ABB RobotStudio station: EstacionTaladrado_20230526-132759.rsstn

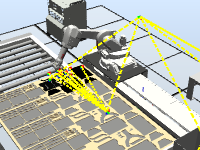
Station EstacionTaladrado (saved by RobotStudio 6.8.8307.1040)
Controller IRB1600APM, task T_ROB2: task frame (RAPID world) sits at (108, -1423.5, 460) mm, rotated rx 0 ry 0 rz 90 deg in the station
Controller IRB1600APM, task T_ROB1: task frame (RAPID world) sits at (108, -1423.5, 460) mm, rotated rx 0 ry 0 rz 90 deg in the station
Controller IRB1600APM
  mechanical unit ROB_1: IRB1600_6_145_A, 6 joints, base frame (0, 0, 0) mm
  mechanical unit TRACK_1: IRBT2005_IRB_STD_INT_0_0_4_A, 1 joints, base frame (0, 0, 0) mm
  mechanical unit ROB_2: IRB1600_6_145_B, 6 joints, base frame (1847, 2866, 0) mm, rotated rx 0 ry 0 rz 180 deg
  mechanical unit TRACK_2: IRBT2005_IRB_STD_INT_0_0_4_B, 1 joints, base frame (1847, 2866, 0) mm, rotated rx 0 ry 0 rz 180 deg
Layout (positions relative to the parent item):
  - Placa_de_Corte [part] at (-2250, -1220, 450) mm
  - IRC5_Singel-Cabinet [part, from Equipment\IRC5_Singel-Cabinet.rslib] at (500, 3000, 100) mm, rotated rx 90 ry 0 rz 90 deg
  - 1320_4000_h2 [part, from Equipment\Conveyor 1320 4000 h2.rslib] at (-1985, 2800, 0) mm, rotated rx 0 ry 0 rz -90 deg
  - Ventosa_Smart [smart component]
      signals: DI StartAttacher, DO Executed
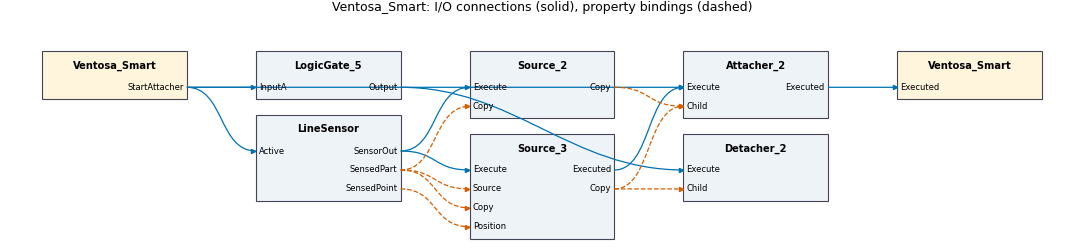
      connections:
        Ventosa_Smart.StartAttacher -> LogicGate_5.InputA
        LogicGate_5.Output -> Detacher_2.Execute
        Ventosa_Smart.StartAttacher -> LineSensor.Active
        Ventosa_Smart.StartAttacher -> Attacher_2.Execute
        Attacher_2.Executed -> Ventosa_Smart.Executed
        LineSensor.SensorOut -> Source_2.Execute
        LineSensor.SensorOut -> Source_3.Execute
        Source_3.Executed -> Attacher_2.Execute
        LineSensor.SensedPart => Source_2.Copy
        Source_2.Copy => Attacher_2.Child
        LineSensor.SensedPart => Source_3.Source
        LineSensor.SensedPart => Source_3.Copy
        Source_3.Copy => Attacher_2.Child
        Source_3.Copy => Detacher_2.Child
        LineSensor.SensedPoint => Source_3.Position
    - Attacher_2 [smart component, from Components\Attacher.rslib]
        properties: Parent=Ventosa; Flange=0; Child=(none); Mount=false; Offset=[0 0 0]; Orientation=[0 0 0]
    - Detacher_2 [smart component, from Components\Detacher.rslib]
        properties: Child=(none); KeepPosition=true
    - LogicGate_5 [smart component, from Components\LogicGate.rslib]
        properties: Operator=NOT; Delay=0
    - LineSensor [smart component, from Components\LineSensor.rslib] at (-959.44, 1157.84, 473.42) mm, rotated rx -180 ry 0 rz 0 deg
        properties: Start=[0 0 0]; End=[6.66133814775094E-16 -4.71844785465692E-16 0.00999998807907376]; Radius=0.006; SensedPart=(none); SensedPoint=[0 0 0]
      - _sensorPart_ [part]
    - Ventosa [mechanism, from Libraries\Ventosa.rslib] at (-959.44, 1157.84, 583.42) mm, rotated rx -180 ry 0 rz 0 deg
    - Source_3 [smart component, from Components\Source.rslib]
        properties: Source=(none); Copy=(none); Parent=(none); Position=[0 0 0]; Orientation=[0 0 0]; Transient=false; PhysicsBehavior=0
  - PLACA_SOPORTE_1 [part] at (-1200.46, 988.98, 450) mm
  - BANDEJA_LAMINA [part]
  - MyTool [mechanism, from Training Objects\myTool.rslib] at (-2758, -382.79, 1614) mm, rotated rx 180 ry 60 rz 90 deg
  - SOPORTE_LATERAL_SOPORTE_1 [part] at (-961.81, 1075.54, 450) mm
  - MESA_TALADRADO [part] at (1200, -425, 400) mm
  - MESA_TALADRADO_B [part] at (-3850, 0, 400) mm
  - IRB1600_6_145_A [mechanism, from Robots\IRB1600_6_145_G_02.rslib] at (108, 926.5, 460) mm, rotated rx 0 ry 0 rz 90 deg; joint values [1.3574, 1.2334, -0.1513, 0, 0.4887, -0.2134] (rad or m)
  - IRB1600_6_145_B [mechanism, from Robots\IRB1600_6_145_G_02.rslib] at (-2758, 423.5, 460) mm, rotated rx 0 ry 0 rz -90 deg; joint values [0, 0, 0, 0, 0.5236, 0] (rad or m)
  - IRBT2005_IRB_STD_INT_0_0_4_A [mechanism] at (400, -2248, 0) mm, rotated rx 0 ry 0 rz 90 deg; joint values [2.35] (rad or m)
      links: Base, Link1
  - IRBT2005_IRB_STD_INT_0_0_4_B [mechanism] at (-3050, 1248, 0) mm, rotated rx 0 ry 0 rz -90 deg; joint values [0] (rad or m)
      links: Base, Link1
  - Conveyor_A [smart component]
      signals: DI MoveConv
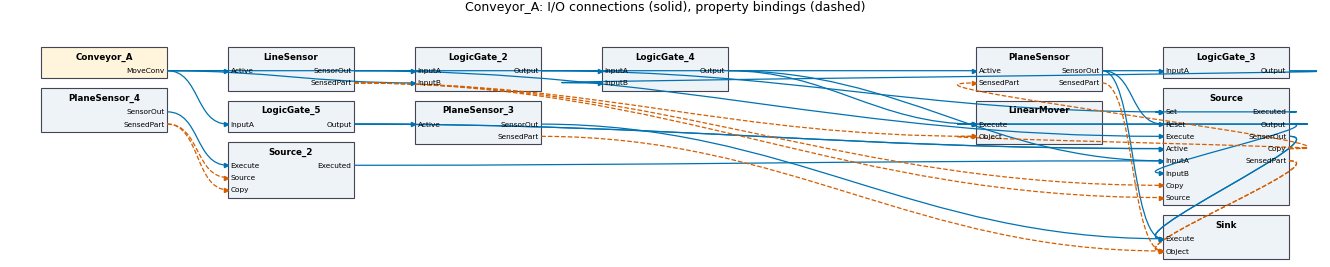
      connections:
        Source.Executed -> LogicSRLatch.Set
        PlaneSensor.SensorOut -> LogicSRLatch.Reset
        Conveyor_A.MoveConv -> LineSensor.Active
        LineSensor.SensorOut -> Source.Execute
        LogicSRLatch.Output -> LinearMover.Execute
        Conveyor_A.MoveConv -> PlaneSensor.Active
        LineSensor.SensorOut -> LogicGate_2.InputA
        Conveyor_A.MoveConv -> LogicGate_2.InputB
        LogicGate_2.Output -> LogicSRLatch.Set
        PlaneSensor.SensorOut -> LogicGate_3.InputA
        LogicGate_2.Output -> LogicGate_4.InputA
        LogicGate_3.Output -> LogicGate_4.InputB
        PlaneSensor.SensorOut -> Sink.Execute
        PlaneSensor_2.SensorOut -> Sink.Execute
        Conveyor_A.MoveConv -> LogicGate_5.InputA
        LogicGate_5.Output -> PlaneSensor_2.Active
        LogicGate_5.Output -> LineSensor.Active
        LineSensor.SensorOut -> Sink.Execute
        PlaneSensor_3.SensorOut -> Sink.Execute
        LogicGate_5.Output -> PlaneSensor_3.Active
        PlaneSensor_4.SensorOut -> Source_2.Execute
        LogicGate_4.Output -> LogicGate_8.InputA
        LogicGate_8.Output -> LinearMover.Execute
        LogicGate_9.Output -> LogicGate_8.InputB
        Source_2.Executed -> LogicGate_9.InputA
        LogicGate_4.Output -> LinearMover.Execute
        LineSensor.SensedPart => Source.Copy
        Source.Copy => LinearMover.Object
        Source.Copy => PlaneSensor.SensedPart
        LineSensor.SensedPart => Source.Source
        PlaneSensor_2.SensedPart => Sink.Object
        LineSensor.SensedPart => Sink.Object
        PlaneSensor_3.SensedPart => Sink.Object
        LineSensor.SensedPart => LinearMover.Object
        PlaneSensor.SensedPart => Sink.Object
        PlaneSensor_4.SensedPart => Source_2.Source
        PlaneSensor_4.SensedPart => Source_2.Copy
    - PlaneSensor [smart component, from Components\PlaneSensor.rslib]
        properties: Origin=[-1.025 -4.3 0.776]; Axis1=[0 0 0.099]; Axis2=[0.39 0 0]; SensedPart=(none)
      - _sensorPart_ [part]
    - LineSensor [smart component, from Components\LineSensor.rslib]
        properties: Start=[-0.83 -1.7 0.78]; End=[-0.83 -4.3 0.785]; Radius=0.005; SensedPart=BOX_A; SensedPoint=[-0.83 -1.7 0.78]
      - _sensorPart_ [part]
    - LinearMover [smart component, from Components\LinearMover.rslib]
        properties: Object=BOX_A; Direction=[0 -3.5 0]; Speed=0.5; Reference=Global; ReferenceObject=(none)
    - LogicGate_2 [smart component, from Components\LogicGate.rslib]
        properties: Operator=AND; Delay=0
    - LogicGate_3 [smart component, from Components\LogicGate.rslib]
        properties: Operator=NOT; Delay=0
    - LogicGate_4 [smart component, from Components\LogicGate.rslib]
        properties: Operator=AND; Delay=0
    - Sink [smart component, from Components\Sink.rslib]
        properties: Object=(none)
    - LogicGate_5 [smart component, from Components\LogicGate.rslib]
        properties: Operator=NOT; Delay=0
    - PlaneSensor_3 [smart component, from Components\PlaneSensor.rslib]
        properties: Origin=[-1.02 -2 0.786]; Axis1=[0.38 0 0]; Axis2=[0 0.3 0]; SensedPart=(none)
      - _sensorPart_ [part]
    - Source_2 [smart component, from Components\Source.rslib]
        properties: Source=(none); Copy=(none); Parent=(none); Position=[-0.83 -1.85 0.776]; Orientation=[0 0 0]; Transient=false; PhysicsBehavior=0
    - PlaneSensor_4 [smart component, from Components\PlaneSensor.rslib]
        properties: Origin=[-1.025 -4.3 0.776]; Axis1=[0 0 0.099]; Axis2=[0.39 0 0]; SensedPart=(none)
      - _sensorPart_ [part]
  - 400_guide_B [part, from Equipment\Conveyor Guide 400.rslib] at (-1955, -1500, 0) mm, rotated rx 0 ry 0 rz -90 deg
  - 400_guide_A [part, from Equipment\Conveyor Guide 400.rslib] at (-1030, -1500, 0) mm, rotated rx 0 ry 0 rz -90 deg
  - SOPORTE_LATERAL_SOPORTE_1_2 [part] at (-1011.44, 1038.99, 450) mm
  - BASE_SOPORTE_1 [part] at (-878.76, 996.15, 450) mm
  - GRADUADOR_INCLINACION_SOPORTE_1 [part] at (-1023.59, 997.95, 450) mm
  - GRADUADOR_INCLINACION_SOPORTE_1_2 [part] at (-966.4, 1160.33, 450) mm
  - SUJECION_CENTRAL_SOPORTE_1 [part] at (-870.47, 885.99, 450) mm
  - BRAZO_SOPORTE_1 [part] at (-762.24, 1077.84, 450) mm
  - BRAZO_2_SOPORTE_1 [part] at (-1135.46, 1150.12, 450) mm
  - BOX_A [part] at (-830, -1850, 776) mm
  - PLACA_INFERIOR_MESA_1 [part] at (-558.01, 1007.22, 450) mm
  - PLACA_SUPERIOR_MESA_1 [part] at (-913.92, 730.48, 450) mm
  - SOPORTE_LATERAL_I_MESA_1 [part] at (-1245.6, 782.8, 450) mm
  - SOPORTE_LATERAL_D_MESA_1 [part] at (-580.16, 719.3, 450) mm
Attachment: LineSensor is attached to Ventosa / HERRAMIENTA
Attachment: Ventosa is attached to IRB1600_6_145_A / Link6
Attachment: MyTool is attached to IRB1600_6_145_B / Link6
Attachment: IRB1600_6_145_A is attached to IRBT2005_IRB_STD_INT_0_0_4_A / Link1
Attachment: IRB1600_6_145_B is attached to IRBT2005_IRB_STD_INT_0_0_4_B / Link1
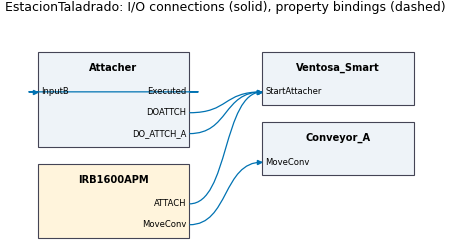
Station logic (signal -> signal, property => property):
  Attacher.Executed -> LogicGate.InputB
  IRB1600APM.DOATTCH -> Ventosa_Smart.StartAttacher
  IRB1600APMSYS.DO_ATTCH_A -> Ventosa_Smart.StartAttacher
  IRB1600APM.ATTACH -> Ventosa_Smart.StartAttacher
  IRB1600APM.MoveConv -> Conveyor_A.MoveConv
Targets, tools, work objects and paths stored in the station, written as RAPID:
! task T_ROB1
MODULE CalibData
  PERS tooldata VentosaTCP:=[TRUE,[[0,0,110.772],[1,0,0,0]],[1,[0,0,53.582],[1,0,0,0],0,0,0]];
  TASK PERS wobjdata PLACA_A:=[FALSE,TRUE,"",[[0,0,0],[1,0,0,0]],[[203.5,2358,-10],[0.707106781,0,0,-0.707106781]]];
ENDMODULE

! task T_ROB1
MODULE Module1
  CONST jointtarget HOME_A:=[[0,0,0,0,30,0],[925,9E+09,9E+09,9E+09,9E+09,9E+09]];
  CONST jointtarget MID_A:=[[90,60,-20,0,50,0],[925,9E+09,9E+09,9E+09,9E+09,9E+09]];
  CONST jointtarget TABLE_A:=[[-86.149,71.536,-9.408,0,27.873,0],[925,9E+09,9E+09,9E+09,9E+09,9E+09]];
  CONST jointtarget SLS1_A:=[[82.069,70.996,-7.558,0,26.562,0],[2350,9E+09,9E+09,9E+09,9E+09,9E+09]];
  CONST jointtarget PS1_A:=[[87.22,84.052,-44.6,0,50.548,0],[2349.769019747,9E+09,9E+09,9E+09,9E+09,9E+09]];
  CONST jointtarget PS1_AA:=[[87.22,83.446,-44.115,0,50.669,0],[2349.769019747,9E+09,9E+09,9E+09,9E+09,9E+09]];
  CONST jointtarget PSLS1_AA:=[[82.069,69.527,-6.738,0,27.211,0],[2350,9E+09,9E+09,9E+09,9E+09,9E+09]];
  CONST jointtarget CONVEYOR_A:=[[84.914,41.92,15.328,-0.622,32.813,0],[-461.181385797,9E+09,9E+09,9E+09,9E+09,9E+09]];
  CONST jointtarget MID_CONV_A:=[[89.175,20.381,4.444,0.004,65.253,0],[-480,9E+09,9E+09,9E+09,9E+09,9E+09]];
  CONST jointtarget SLS12_AA:=[[84.262,72.054,-13.066,0,31.013,0],[2350,9E+09,9E+09,9E+09,9E+09,9E+09]];
  CONST jointtarget SLS12_A:=[[84.105,72.802,-13.543,0,30.74,0],[2350,9E+09,9E+09,9E+09,9E+09,9E+09]];
  CONST jointtarget BS1_A:=[[84.635,68.196,3.223,0,18.581,0],[2350,9E+09,9E+09,9E+09,9E+09,9E+09]];
  CONST jointtarget BS1_AA:=[[84.635,67.383,3.658,0,18.96,0],[2350,9E+09,9E+09,9E+09,9E+09,9E+09]];
  CONST jointtarget GIS1_AA:=[[86.51,72.134,-13.296,0,31.162,0],[2350,9E+09,9E+09,9E+09,9E+09,9E+09]];
  CONST jointtarget GIS1_A:=[[86.51,72.86,-13.724,0,30.865,0],[2350,9E+09,9E+09,9E+09,9E+09,9E+09]];
  CONST jointtarget GIS12_AA:=[[77.771,70.671,-8.671,0,28,0],[2350,9E+09,9E+09,9E+09,9E+09,9E+09]];
  CONST jointtarget GIS12_A:=[[77.79,71.449,-9.107,0,27.659,0],[2350,9E+09,9E+09,9E+09,9E+09,9E+09]];
  CONST jointtarget BRS1_A:=[[80.135,66.069,14.969,0,8.962,0],[2350,9E+09,9E+09,9E+09,9E+09,9E+09]];
  CONST jointtarget BRS1_AA:=[[80.135,65.237,15.395,0,9.368,0],[2350,9E+09,9E+09,9E+09,9E+09,9E+09]];
  CONST jointtarget BRS12_A:=[[79.805,80.411,-35.266,0,44.855,0],[2350,9E+09,9E+09,9E+09,9E+09,9E+09]];
  CONST jointtarget BRS12_AA:=[[79.805,79.69,-34.75,0,45.061,0],[2350,9E+09,9E+09,9E+09,9E+09,9E+09]];
  CONST jointtarget SCS1_A:=[[92.371,67.896,4.57,0,17.533,0],[2350,9E+09,9E+09,9E+09,9E+09,9E+09]];
  CONST jointtarget SCS1_AA:=[[92.371,67.108,4.99,0,17.903,0],[2350,9E+09,9E+09,9E+09,9E+09,9E+09]];
  CONST jointtarget PIM1_A:=[[56.022,65.432,22.991,0,1.578,0],[1981.865508797,9E+09,9E+09,9E+09,9E+09,9E+09]];
  CONST jointtarget PIM1_AA:=[[56.022,64.534,23.445,0,2.021,0],[1981.865508797,9E+09,9E+09,9E+09,9E+09,9E+09]];
  CONST jointtarget TABLE_AA:=[[-86.149,55.011,-3.204,0,38.193,0],[925,9E+09,9E+09,9E+09,9E+09,9E+09]];
  CONST jointtarget TABLE_A90:=[[-86.149,55.011,-3.204,0,38.193,90],[925,9E+09,9E+09,9E+09,9E+09,9E+09]];
  CONST jointtarget TABLE_A180:=[[-86.149,55.011,-3.204,0,38.193,180],[925,9E+09,9E+09,9E+09,9E+09,9E+09]];
  CONST jointtarget TABLE_A270:=[[-86.149,55.011,-3.204,0,38.193,270],[925,9E+09,9E+09,9E+09,9E+09,9E+09]];
  PROC Path_HOME_A()
    MoveAbsJ HOME_A,v1000,z100,VentosaTCP\WObj:=PLACA_A;
  ENDPROC
  PROC Path_MID_A()
    MoveAbsJ MID_A,v1000,z100,VentosaTCP\WObj:=PLACA_A;
  ENDPROC
  PROC Path_PS1_A()
    MoveAbsJ PS1_A,v1000,z100,VentosaTCP\WObj:=PLACA_A;
    MoveAbsJ PS1_AA,v1000,z100,VentosaTCP\WObj:=PLACA_A;
    MoveAbsJ HOME_A,v1000,z100,VentosaTCP\WObj:=PLACA_A;
    MoveAbsJ MID_CONV_A,v1000,z100,VentosaTCP\WObj:=PLACA_A;
    MoveAbsJ CONVEYOR_A,v1000,z100,VentosaTCP\WObj:=PLACA_A;
  ENDPROC
  PROC Path_PS1_AA()
    MoveAbsJ PS1_AA,v1000,z100,VentosaTCP\WObj:=PLACA_A;
  ENDPROC
  PROC Path_MID_CONV_A()
    MoveAbsJ MID_CONV_A,v1000,z100,VentosaTCP\WObj:=PLACA_A;
  ENDPROC
  PROC Path_SLS1_A()
    MoveAbsJ SLS1_A,v1000,z100,VentosaTCP\WObj:=PLACA_A;
    MoveAbsJ PSLS1_AA,v1000,z100,VentosaTCP\WObj:=PLACA_A;
    MoveAbsJ MID_A,v1000,z100,VentosaTCP\WObj:=PLACA_A;
    MoveAbsJ HOME_A,v1000,z100,VentosaTCP\WObj:=PLACA_A;
    MoveAbsJ TABLE_A,v1000,z100,VentosaTCP\WObj:=PLACA_A;
  ENDPROC
  PROC Path_SLS1_AA()
    MoveAbsJ PSLS1_AA,v1000,z100,VentosaTCP\WObj:=PLACA_A;
  ENDPROC
  PROC Path_SLS12_AA()
    MoveAbsJ SLS12_AA,v1000,z100,VentosaTCP\WObj:=PLACA_A;
  ENDPROC
  PROC Path_SLS12_A()
    MoveAbsJ SLS12_A,v1000,z100,VentosaTCP\WObj:=PLACA_A;
    MoveAbsJ SLS12_AA,v1000,z100,VentosaTCP\WObj:=PLACA_A;
    MoveAbsJ MID_A,v1000,z100,VentosaTCP\WObj:=PLACA_A;
    MoveAbsJ HOME_A,v1000,z100,VentosaTCP\WObj:=PLACA_A;
    MoveAbsJ TABLE_A,v1000,z100,VentosaTCP\WObj:=PLACA_A;
  ENDPROC
  PROC Path_BS1_A()
    MoveAbsJ BS1_A,v1000,z10,VentosaTCP\WObj:=PLACA_A;
    MoveAbsJ BS1_AA,v1000,z10,VentosaTCP\WObj:=PLACA_A;
    MoveAbsJ MID_A,v1000,z10,VentosaTCP\WObj:=PLACA_A;
    MoveAbsJ HOME_A,v1000,z10,VentosaTCP\WObj:=PLACA_A;
    MoveAbsJ MID_CONV_A,v1000,z10,VentosaTCP\WObj:=PLACA_A;
    MoveAbsJ CONVEYOR_A,v1000,z10,VentosaTCP\WObj:=PLACA_A;
  ENDPROC
  PROC Path_BS1_AA()
    MoveAbsJ BS1_AA,v1000,z10,VentosaTCP\WObj:=PLACA_A;
  ENDPROC
  PROC Path_SLS1_A_2()
    MoveAbsJ HOME_A,v1000,z100,VentosaTCP\WObj:=PLACA_A;
    MoveAbsJ MID_CONV_A,v1000,z100,VentosaTCP\WObj:=PLACA_A;
    MoveAbsJ CONVEYOR_A,v1000,z100,VentosaTCP\WObj:=PLACA_A;
  ENDPROC
  PROC Path_SLS12_A_2()
    MoveAbsJ HOME_A,v1000,z100,VentosaTCP\WObj:=PLACA_A;
    MoveAbsJ MID_CONV_A,v1000,z100,VentosaTCP\WObj:=PLACA_A;
    MoveAbsJ CONVEYOR_A,v1000,z100,VentosaTCP\WObj:=PLACA_A;
  ENDPROC
  PROC Path_GIS1_A()
    MoveAbsJ GIS1_A,v1000,z10,VentosaTCP\WObj:=PLACA_A;
    MoveAbsJ GIS1_AA,v1000,z10,VentosaTCP\WObj:=PLACA_A;
    MoveAbsJ MID_A,v1000,z10,VentosaTCP\WObj:=PLACA_A;
    MoveAbsJ HOME_A,v1000,z10,VentosaTCP\WObj:=PLACA_A;
    MoveAbsJ TABLE_A,v1000,z10,VentosaTCP\WObj:=PLACA_A;
  ENDPROC
  PROC Path_GIS1_AA()
    MoveAbsJ GIS1_AA,v1000,z10,VentosaTCP\WObj:=PLACA_A;
  ENDPROC
  PROC Path_GIS1_A_2()
    MoveAbsJ HOME_A,v1000,z10,VentosaTCP\WObj:=PLACA_A;
    MoveAbsJ MID_CONV_A,v1000,z10,VentosaTCP\WObj:=PLACA_A;
    MoveAbsJ CONVEYOR_A,v1000,z10,VentosaTCP\WObj:=PLACA_A;
  ENDPROC
  PROC Path_GIS12_AA()
    MoveAbsJ GIS12_AA,v1000,z10,VentosaTCP\WObj:=PLACA_A;
  ENDPROC
  PROC Path_GIS12_A()
    MoveAbsJ GIS12_A,v1000,z10,VentosaTCP\WObj:=PLACA_A;
    MoveAbsJ GIS12_AA,v1000,z10,VentosaTCP\WObj:=PLACA_A;
    MoveAbsJ MID_A,v1000,z10,VentosaTCP\WObj:=PLACA_A;
    MoveAbsJ HOME_A,v1000,z10,VentosaTCP\WObj:=PLACA_A;
    MoveAbsJ TABLE_A,v1000,z10,VentosaTCP\WObj:=PLACA_A;
  ENDPROC
  PROC Path_GIS12_A_2()
    MoveAbsJ HOME_A,v1000,z10,VentosaTCP\WObj:=PLACA_A;
    MoveAbsJ MID_CONV_A,v1000,z10,VentosaTCP\WObj:=PLACA_A;
    MoveAbsJ CONVEYOR_A,v1000,z10,VentosaTCP\WObj:=PLACA_A;
  ENDPROC
  PROC Path_BRS1_A()
    MoveAbsJ BRS1_A,v1000,z10,VentosaTCP\WObj:=PLACA_A;
    MoveAbsJ BRS1_AA,v1000,z10,VentosaTCP\WObj:=PLACA_A;
    MoveAbsJ MID_A,v1000,z10,VentosaTCP\WObj:=PLACA_A;
    MoveAbsJ HOME_A,v1000,z10,VentosaTCP\WObj:=PLACA_A;
    MoveAbsJ MID_CONV_A,v1000,z10,VentosaTCP\WObj:=PLACA_A;
    MoveAbsJ CONVEYOR_A,v1000,z10,VentosaTCP\WObj:=PLACA_A;
  ENDPROC
  PROC Path_BRS1_AA()
    MoveAbsJ BRS1_AA,v1000,z10,VentosaTCP\WObj:=PLACA_A;
  ENDPROC
  PROC Path_BRS12_A()
    MoveAbsJ BRS12_A,v1000,z10,VentosaTCP\WObj:=PLACA_A;
    MoveAbsJ BRS12_AA,v1000,z10,VentosaTCP\WObj:=PLACA_A;
    MoveAbsJ MID_A,v1000,z10,VentosaTCP\WObj:=PLACA_A;
    MoveAbsJ HOME_A,v1000,z10,VentosaTCP\WObj:=PLACA_A;
    MoveAbsJ MID_CONV_A,v1000,z10,VentosaTCP\WObj:=PLACA_A;
    MoveAbsJ CONVEYOR_A,v1000,z10,VentosaTCP\WObj:=PLACA_A;
  ENDPROC
  PROC Path_BRS12_AA()
    MoveAbsJ BRS12_AA,v1000,z10,VentosaTCP\WObj:=PLACA_A;
  ENDPROC
  PROC Path_SCS1_A()
    MoveAbsJ SCS1_A,v1000,z10,VentosaTCP\WObj:=PLACA_A;
    MoveAbsJ SCS1_AA,v1000,z10,VentosaTCP\WObj:=PLACA_A;
    MoveAbsJ MID_A,v1000,z10,VentosaTCP\WObj:=PLACA_A;
    MoveAbsJ HOME_A,v1000,z10,VentosaTCP\WObj:=PLACA_A;
    MoveAbsJ TABLE_A,v1000,z10,VentosaTCP\WObj:=PLACA_A;
  ENDPROC
  PROC Path_SCS1_AA()
    MoveAbsJ SCS1_AA,v1000,z10,VentosaTCP\WObj:=PLACA_A;
  ENDPROC
  PROC Path_SCS1_A_2()
    MoveAbsJ HOME_A,v1000,z10,VentosaTCP\WObj:=PLACA_A;
    MoveAbsJ MID_CONV_A,v1000,z10,VentosaTCP\WObj:=PLACA_A;
    MoveAbsJ CONVEYOR_A,v1000,z10,VentosaTCP\WObj:=PLACA_A;
  ENDPROC
  PROC Path_PIM1_A()
    MoveAbsJ PIM1_A,v1000,z10,VentosaTCP\WObj:=PLACA_A;
    MoveAbsJ PIM1_AA,v1000,z10,VentosaTCP\WObj:=PLACA_A;
    MoveAbsJ MID_A,v1000,z10,VentosaTCP\WObj:=PLACA_A;
    MoveAbsJ HOME_A,v1000,z10,VentosaTCP\WObj:=PLACA_A;
    MoveAbsJ TABLE_AA,v1000,z10,VentosaTCP\WObj:=PLACA_A;
    MoveAbsJ TABLE_A,v1000,z10,VentosaTCP\WObj:=PLACA_A;
  ENDPROC
  PROC Path_PIM1_AA()
    MoveAbsJ PIM1_AA,v1000,z10,VentosaTCP\WObj:=PLACA_A;
  ENDPROC
  PROC Path_PIM1_A_2()
    MoveAbsJ TABLE_AA,v1000,z10,VentosaTCP\WObj:=PLACA_A;
    MoveAbsJ TABLE_A90,v1000,z10,VentosaTCP\WObj:=PLACA_A;
  ENDPROC
  PROC Path_PIM1_A_3()
    MoveAbsJ TABLE_AA,v1000,z10,VentosaTCP\WObj:=PLACA_A;
    MoveAbsJ TABLE_A180,v1000,z10,VentosaTCP\WObj:=PLACA_A;
  ENDPROC
  PROC Path_PIM1_A_4()
    MoveAbsJ TABLE_AA,v1000,z10,VentosaTCP\WObj:=PLACA_A;
    MoveAbsJ TABLE_A270,v1000,z10,VentosaTCP\WObj:=PLACA_A;
  ENDPROC
  PROC Path_PIM1_A_5()
    MoveAbsJ TABLE_AA,v1000,z10,VentosaTCP\WObj:=PLACA_A;
    MoveAbsJ HOME_A,v1000,z10,VentosaTCP\WObj:=PLACA_A;
    MoveAbsJ MID_CONV_A,v1000,z10,VentosaTCP\WObj:=PLACA_A;
    MoveAbsJ CONVEYOR_A,v1000,z10,VentosaTCP\WObj:=PLACA_A;
  ENDPROC
ENDMODULE

! task T_ROB2
MODULE CalibData
  PERS tooldata MyTool:=[TRUE,[[31.792631019,0,229.638935148],[0.945518576,0,0.325568154,0]],[1,[0,0,1],[1,0,0,0],0,0,0]];
ENDMODULE

